FUNCTION_BLOCK EvetLogger
VAR
	EventBuffer : ARRAY [1..MaxNumberOfArray] OF ST_Events;
	CurrentBufferEntry : INT := 1;
END_VAR
VAR CONSTANT
	MaxNumberOfArray : INT := 100;
END_VAR

METHOD PUBLIC AddEvent : BOOL
VAR_INPUT
	eEventType : E_EventType;
	eEventSeverity : TcEventSeverity;
	eEventIdentity : UDINT;
	eEventText : STRING(255);
END_VAR
IF NOT IsBufferFull() THEN
	CurrentBufferEntry := CurrentBufferEntry +1 ;
	EventBuffer [CurrentBufferEntry].eEventType := eEventType;
	EventBuffer [CurrentBufferEntry].eEventIdentity := eEventIdentity;
	EventBuffer [CurrentBufferEntry].eEventSeverity := eEventSeverity;
	EventBuffer [CurrentBufferEntry].eEventText := eEventText;
	FUpdateEventTimeStampedWithSystemTimeStamepd(EventBuffer [CurrentBufferEntry]);
	AddEvent := TRUE;
ELSE 
	AddEvent := FALSE;
END_IF
END_METHOD

METHOD PUBLIC IsBufferFull : BOOL
VAR_INPUT
END_VAR
IF (CurrentBufferEntry + 1) > MaxNumberOfArray THEN
	IsBufferFull := TRUE;
ELSE 
	IsBufferFull := FALSE;
END_IF
END_METHOD

END_FUNCTION_BLOCK

(* stored: Version 1.1.0.1, ProductVersion 3.1.4024.12
   POU EvetLogger: Id {ec2493a7-1fbe-48bd-880f-1b243969ed21}, SpecialFunc None
   Method AddEvent: Id {076bde83-de45-4a65-b1f5-bf50b435044c}
   Method IsBufferFull: Id {244cae99-4afa-410e-b1be-9449ca8ea731} *)
